// ------------------------------------------------------------------ //
// Section 0 -- cursor baseline, and the enable/disable edges.
// ------------------------------------------------------------------ //

// First time we ever run, adopt whatever the ring can still supply rather than
// starting at nWriteIdx. Someone who enables logging after noticing trouble
// wants the entries that are still there, not only the ones from now on. Bounded
// by RING because older slots have already been overwritten.
IF NOT bCursorSet THEN
    bCursorSet := TRUE;
    IF GVL_Log.nWriteIdx > RING THEN
        udiLastRead := GVL_Log.nWriteIdx - RING;
    ELSE
        udiLastRead := 0;
    END_IF
END_IF

// Turning logging OFF must not abandon a part-written flush or a full buffer:
// drain what is pending and close cleanly, THEN go idle.
fbTrigOff(CLK := NOT GVL_HmiPersistent.stLogFileCfg.bEnabled);
IF fbTrigOff.Q AND (GVL_Log.nWriteIdx > udiLastRead) THEN
    bClosing := TRUE;
END_IF

udiPending := GVL_Log.nWriteIdx - udiLastRead;

// ------------------------------------------------------------------ //
// Section 1 -- flush trigger.
//
// The quiet timer is the flash-wear control: entries collect in the ring and
// reach the card once per uiFlushSec, so a busy second costs one open/close
// rather than dozens. HIGH_WATER is the safety valve -- at 200 of 256 pending
// we stop waiting for the timer, because passing 256 loses entries.
// ------------------------------------------------------------------ //
tonFlush(IN  := (udiPending > 0) AND GVL_HmiPersistent.stLogFileCfg.bEnabled,
         PT  := UDINT_TO_TIME(GVL_HmiPersistent.stLogFileCfg.uiFlushSec * 1000));

// ------------------------------------------------------------------ //
// Section 2 -- the state machine.
// ------------------------------------------------------------------ //
CASE eStep OF

// ---------------- 0: idle ---------------- //
0:
    // OFF means "not logging". BUFFER means "logging, entries accumulating in the
    // ring, waiting for the flush interval". Reporting OFF while enabled would
    // read as a fault on the Logs page when nothing is wrong.
    IF GVL_HmiPersistent.stLogFileCfg.bEnabled THEN
        GVL_Log.stLogFile.eState := E_LogFileState.BUFFER;
    ELSE
        GVL_Log.stLogFile.eState := E_LogFileState.OFF;
    END_IF

    IF (GVL_HmiPersistent.stLogFileCfg.bEnabled OR bClosing)
       AND (udiPending > 0)
       AND (tonFlush.Q OR (udiPending >= HIGH_WATER) OR bClosing) THEN

        // OVERFLOW CHECK, before anything else touches the cursor. If more than
        // RING entries arrived since we last read, the oldest are already
        // overwritten and are gone -- unavoidable, the ring is finite. What is
        // NOT acceptable is losing them silently, so the count is published AND
        // a synthetic row goes into the file itself. A reader of the CSV must be
        // able to see the gap without also having to read a PLC symbol.
        IF udiPending > RING THEN
            udiLostNow := udiPending - RING;
            GVL_Log.stLogFile.udiEntriesDropped :=
                GVL_Log.stLogFile.udiEntriesDropped + udiLostNow;
            udiLastRead := GVL_Log.nWriteIdx - RING;
            bLossRow    := TRUE;
        END_IF

        GVL_Log.stLogFile.eState := E_LogFileState.BUFFER;
        eStep := 5;
    END_IF

// ---------------- 5: make sure the directory exists ---------------- //
// Once per session. Errors are IGNORED on purpose: "already exists" is an error
// from this FB and is also the normal case, and distinguishing it from a real
// failure by error number would be guessing. If the directory genuinely cannot
// be made, the open in state 20 fails and THAT is reported -- one authoritative
// error rather than two competing ones.
5:
    IF bDirTried THEN
        eStep := 10;
    ELSE
        sDirNoSlash := GVL_HmiPersistent.stLogFileCfg.sDir;
        IF (LEN(sDirNoSlash) > 1)
           AND (RIGHT(sDirNoSlash, 1) = '\') THEN
            sDirNoSlash := LEFT(sDirNoSlash, LEN(sDirNoSlash) - 1);
        END_IF
        fbMkDir(sPathName := sDirNoSlash,
                ePath     := Tc2_System.PATH_GENERIC,
                bExecute  := TRUE,
                tTimeout  := FILE_TO);
        IF NOT fbMkDir.bBusy THEN
            fbMkDir(bExecute := FALSE);
            bDirTried := TRUE;
            eStep := 10;
        END_IF
    END_IF

// ---------------- 10: filename, and does it already exist? ---------------- //
10:
    IF GVL_Log.sToday = '0000-00-00' THEN
        // The panel RTC is unset. Naming a file from that would produce
        // something like flower-0000-00-00.csv, which sorts before every real
        // file and would be deleted first by the Phase 3 retention sweep -- so
        // the one file written while the clock was broken would be the first to
        // go. A distinct name keeps it identifiable and out of the date order.
        sFileName := 'flower-nodate.csv';
    ELSE
        sFileName := CONCAT(CONCAT('flower-', GVL_Log.sToday), '.csv');
    END_IF
    sPath := CONCAT(GVL_HmiPersistent.stLogFileCfg.sDir, sFileName);

    IF sFileName = sLastFile THEN
        bNeedHeader := FALSE;       // same file we appended to last time
        eStep := 20;
    ELSE
        eStep := 11;                // new name -- has to be tested
    END_IF

// ---------------- 11/12: existence probe ---------------- //
// A header belongs at the top of a file, once. Opening in append mode cannot
// tell us whether we created it, so we test first with a READ open: 1804 means
// absent, which is the one error code this project has verified on the panel.
// Costs one extra call per new file, i.e. once a day.
11:
    fbProbe(sPathName := sPath,
            nMode     := Tc2_System.FOPEN_MODEREAD,
            ePath     := Tc2_System.PATH_GENERIC,
            bExecute  := TRUE,
            tTimeout  := FILE_TO);
    IF NOT fbProbe.bBusy THEN
        fbProbe(bExecute := FALSE);
        IF fbProbe.bError THEN
            // Absent -> new file, needs a header. Any OTHER error is left for
            // the append open in state 20 to report, so there is one place that
            // decides the directory is unusable.
            bNeedHeader := (fbProbe.nErrId = E_NOTFOUND);
            eStep := 20;
        ELSE
            bNeedHeader := FALSE;
            hFile := fbProbe.hFile;
            eStep := 12;            // must close the probe handle
        END_IF
    END_IF

12:
    fbClose(hFile := hFile, bExecute := TRUE, tTimeout := FILE_TO);
    IF NOT fbClose.bBusy THEN
        fbClose(bExecute := FALSE);
        hFile := 0;
        eStep := 20;
    END_IF

// ---------------- 20: open for append ---------------- //
20:
    GVL_Log.stLogFile.eState := E_LogFileState.OPENING;
    fbOpen(sPathName := sPath,
           nMode     := Tc2_System.FOPEN_MODEAPPEND OR Tc2_System.FOPEN_MODETEXT,
           ePath     := Tc2_System.PATH_GENERIC,
           bExecute  := TRUE,
           tTimeout  := FILE_TO);
    IF NOT fbOpen.bBusy THEN
        fbOpen(bExecute := FALSE);
        IF fbOpen.bError THEN
            Fail(nErr := fbOpen.nErrId, sWhy := 'open failed');
        ELSE
            hFile := fbOpen.hFile;
            IF bNeedHeader THEN
                sLastFile := sFileName;
                GVL_Log.stLogFile.sCurrentFile := sFileName;
                GVL_Log.stLogFile.uiBytesInFile := 0;
                eStep := 25;
            ELSE
                sLastFile := sFileName;
                GVL_Log.stLogFile.sCurrentFile := sFileName;
                eStep := 30;
            END_IF
        END_IF
    END_IF

// ---------------- 25: header row, new files only ---------------- //
25:
    GVL_Log.stLogFile.eState := E_LogFileState.WRITING;
    fbPuts(hFile := hFile, sLine := CONCAT(HDR, '$N'),
           bExecute := TRUE, tTimeout := FILE_TO);
    IF NOT fbPuts.bBusy THEN
        fbPuts(bExecute := FALSE);
        IF fbPuts.bError THEN
            Fail(nErr := fbPuts.nErrId, sWhy := 'header write failed');
        ELSE
            // +1 because text mode expands the single $N to CRLF on disk.
            GVL_Log.stLogFile.uiBytesInFile :=
                GVL_Log.stLogFile.uiBytesInFile + INT_TO_UDINT(LEN(HDR)) + 2;
            bNeedHeader := FALSE;
            eStep := 30;
        END_IF
    END_IF

// ---------------- 30: the synthetic loss row, if one is owed ---------------- //
30:
    IF NOT bLossRow THEN
        eStep := 31;
    ELSE
        GVL_Log.stLogFile.eState := E_LogFileState.WRITING;
        sRow := CONCAT(CONCAT(Csv(sIn := GVL_Log.sNow), ',"WARN","LogCsv","'),
                CONCAT(UDINT_TO_STRING(udiLostNow),
                       ' entries lost - CSV writer fell behind the ring"$N'));
        fbPuts(hFile := hFile, sLine := sRow,
               bExecute := TRUE, tTimeout := FILE_TO);
        IF NOT fbPuts.bBusy THEN
            fbPuts(bExecute := FALSE);
            IF fbPuts.bError THEN
                Fail(nErr := fbPuts.nErrId, sWhy := 'loss row write failed');
            ELSE
                GVL_Log.stLogFile.uiBytesInFile :=
                    GVL_Log.stLogFile.uiBytesInFile + INT_TO_UDINT(LEN(sRow)) + 1;
                bLossRow := FALSE;
                eStep := 31;
            END_IF
        END_IF
    END_IF

// ---------------- 31: one row per pass until caught up ---------------- //
31:
    IF udiLastRead >= GVL_Log.nWriteIdx THEN
        eStep := 40;
    ELSE
        // Discard DBG without a file call. Unconditional -- independent of
        // GVL_Log.bDebugMode, which still governs the on-screen ring. DBG is the
        // 1 Hz robot keep-alive trace; it would bury the file and burn the card.
        // Bounded per scan so a long DBG run cannot stretch the PlcTask.
        nSkipped := 0;
        WHILE (udiLastRead < GVL_Log.nWriteIdx)
              AND (nSkipped < MAX_SKIP) DO
            nSlot := UDINT_TO_INT(udiLastRead MOD RING);
            IF GVL_Log.aLog[nSlot].eSev = E_LogSev.DBG THEN
                udiLastRead := udiLastRead + 1;
                nSkipped := nSkipped + 1;
            ELSE
                EXIT;
            END_IF
        END_WHILE

        IF udiLastRead >= GVL_Log.nWriteIdx THEN
            eStep := 40;
        ELSE
            GVL_Log.stLogFile.eState := E_LogFileState.WRITING;
            nSlot := UDINT_TO_INT(udiLastRead MOD RING);
            sRow  := RowFor(nSlot := nSlot);
            fbPuts(hFile := hFile, sLine := sRow,
                   bExecute := TRUE, tTimeout := FILE_TO);
            IF NOT fbPuts.bBusy THEN
                fbPuts(bExecute := FALSE);
                IF fbPuts.bError THEN
                    Fail(nErr := fbPuts.nErrId, sWhy := 'row write failed');
                ELSE
                    // Cursor advances ONLY after the write is confirmed. If it
                    // advanced first, a failure here would drop the entry
                    // permanently and invisibly -- the one outcome this whole FB
                    // is arranged to prevent.
                    udiLastRead := udiLastRead + 1;
                    GVL_Log.stLogFile.uiBytesInFile :=
                        GVL_Log.stLogFile.uiBytesInFile + INT_TO_UDINT(LEN(sRow)) + 1;
                END_IF
            END_IF
        END_IF
    END_IF

// ---------------- 40: close ---------------- //
40:
    GVL_Log.stLogFile.eState := E_LogFileState.CLOSING;
    fbClose(hFile := hFile, bExecute := TRUE, tTimeout := FILE_TO);
    IF NOT fbClose.bBusy THEN
        fbClose(bExecute := FALSE);
        IF fbClose.bError THEN
            Fail(nErr := fbClose.nErrId, sWhy := 'close failed');
        ELSE
            hFile := 0;
            // One INFO out, matching the one ERR in. Same discipline as
            // FB_RobotTcpClient's bStateUnanswered: a repeating condition must
            // not be level-logged into a 20-entry ring.
            IF bErrLogged THEN
                bErrLogged := FALSE;
                GVL_Log.stLogFile.iErrorCode := 0;
                GVL_Log.stLogFile.sErrorText := '';
                F_LogEvent(eSev := E_LogSev.INFO, sSource := 'LogCsv',
                           sMsg  := CONCAT('CSV log recovered, writing ',
                                           sFileName));
            END_IF
            tonFlush(IN := FALSE);      // restart the quiet interval
            bClosing := FALSE;
            eStep := 0;
        END_IF
    END_IF

// ---------------- 90: release the handle on the way to FAILED ---------------- //
// Reached only from Fail() and only when a handle is still open. The close result
// is IGNORED: we are already reporting the original error, and replacing it with
// a close error would lose the diagnosis that matters. What we need from here is
// the handle back, not a second opinion.
90:
    GVL_Log.stLogFile.eState := E_LogFileState.CLOSING;
    fbClose(hFile := hFile, bExecute := TRUE, tTimeout := FILE_TO);
    IF NOT fbClose.bBusy THEN
        fbClose(bExecute := FALSE);
        hFile := 0;
        eStep := 99;
    END_IF

// ---------------- 99: failed -- back off, then retry ---------------- //
// Retry on a TIMER, never every scan. A bad sDir or a full card would otherwise
// produce a file call per scan for as long as the machine runs.
99:
    GVL_Log.stLogFile.eState := E_LogFileState.FAILED;
    tonRetry(IN := TRUE, PT := RETRY_TO);
    IF tonRetry.Q THEN
        tonRetry(IN := FALSE);
        bDirTried := FALSE;             // maybe the card came back
        sLastFile := '';                // re-test existence
        eStep := 0;
    END_IF

END_CASE

// ------------------------------------------------------------------ //
// Section 3 -- the STRING mirror of eState.
//
// Required, not decoration: the classic VISU cannot stringify an enum, so a text
// output bound to eState renders the raw number. Every enum in this project
// carries such a mirror for that reason.
// ------------------------------------------------------------------ //
CASE GVL_Log.stLogFile.eState OF
    E_LogFileState.OFF:      GVL_Log.stLogFile.sStateText := 'OFF';
    E_LogFileState.BUFFER:   GVL_Log.stLogFile.sStateText := 'BUFFER';
    E_LogFileState.OPENING:  GVL_Log.stLogFile.sStateText := 'OPENING';
    E_LogFileState.WRITING:  GVL_Log.stLogFile.sStateText := 'WRITING';
    E_LogFileState.CLOSING:  GVL_Log.stLogFile.sStateText := 'CLOSING';
    E_LogFileState.ROTATING: GVL_Log.stLogFile.sStateText := 'ROTATING';
    E_LogFileState.FAILED:   GVL_Log.stLogFile.sStateText := 'FAILED';
ELSE
    GVL_Log.stLogFile.sStateText := '?';
END_CASE

(*
   RFC 4180 quote one field: wrap in double quotes, and double any quote inside.

   NOT theoretical. Robot frames reach log messages as 'SYNC:NAME=VALUE,...' and
   message text already carries commas and parentheses, so an unquoted field
   would split a row into the wrong number of columns and silently corrupt every
   downstream reader. Verified end-to-end on the panel 2026-08-10: a message
   containing both a comma and a doubled quote came back off the card via FTP and
   parsed as one intact field.

   Every field is quoted, including the fixed ones. Uniform rows are easier to
   reason about than rows where quoting depends on content, and the cost is two
   bytes.
*)
METHOD Csv : STRING(200)
VAR_INPUT
    sIn : STRING(80);
END_VAR
VAR
    j    : INT;
    n    : INT;
    sOut : STRING(200);
    c    : STRING(1);
END_VAR
sOut := '"';
n := LEN(sIn);

FOR j := 1 TO n DO
    c := MID(sIn, 1, j);            // MID(str, len, pos) -- one char at j
    IF c = '"' THEN
        sOut := CONCAT(sOut, '""');
    ELSE
        sOut := CONCAT(sOut, c);
    END_IF
END_FOR

Csv := CONCAT(sOut, '"');
END_METHOD

(*
   Build one CSV row from a ring slot, ending in a bare $N.

   Column order matches the HDR constant. Worst case fits: the four source
   fields are STRING(8), STRING(8), STRING(20) and STRING(80), so fully
   quote-doubled they come to 18 + 18 + 42 + 162, plus three commas and the
   newline = 244 of the 255 available.

   $N and NOT $R$N -- FOPEN_MODETEXT already produces CRLF, and doubling it
   gives \r\r\n. See the FB header.
*)
METHOD RowFor : STRING(255)
VAR_INPUT
    nSlot : INT;
END_VAR
RowFor := CONCAT(Csv(sIn := GVL_Log.aLog[nSlot].sTime), ',');
RowFor := CONCAT(RowFor, CONCAT(Csv(sIn := GVL_Log.aLog[nSlot].sSevText), ','));
RowFor := CONCAT(RowFor, CONCAT(Csv(sIn := GVL_Log.aLog[nSlot].sSource), ','));
RowFor := CONCAT(RowFor, CONCAT(Csv(sIn := GVL_Log.aLog[nSlot].sMsg), '$N'));
END_METHOD

(*
   One place that gives up on a flush: latch the error, release the handle, log
   once, and drop into the backoff state.

   THE LOG IS EDGE-GUARDED, and that is the point of centralising this. A full
   card or a bad sDir repeats every retry interval, and level-logging it would
   flush the 20-entry aRecent ring and hide whatever caused the trouble --
   exactly the defect this project already has open against
   FB_RobotTcpClient's connect-failure path. One ERR in, one INFO out on
   recovery (state 40).

   IT DOES NOT CLOSE THE HANDLE ITSELF. An earlier version did, with one
   bExecute TRUE/FALSE pair in the same scan, which starts the close and disarms
   it before it can finish -- so the handle leaks. Harmless once; but a failure
   that repeats every RETRY_TO leaks one every 30 s for as long as the machine
   runs, and exhausting the runtime's handle table would then present as the file
   blocks having stopped working. So a still-open handle routes through state 90,
   which closes it asynchronously and properly before the backoff.
*)
METHOD Fail : BOOL
VAR_INPUT
    nErr : UDINT;
    sWhy : STRING(40);
END_VAR
GVL_Log.stLogFile.iErrorCode := nErr;
GVL_Log.stLogFile.sErrorText :=
    CONCAT(CONCAT(sWhy, ' err '), UDINT_TO_STRING(nErr));

IF NOT bErrLogged THEN
    bErrLogged := TRUE;
    F_LogEvent(eSev := E_LogSev.ERR, sSource := 'LogCsv',
               sMsg  := CONCAT(CONCAT(GVL_Log.stLogFile.sErrorText, ' ('),
                               CONCAT(sPath, ')')));
END_IF

bClosing := FALSE;

// A handle we opened is still open -- close it properly first (state 90) rather
// than abandoning it. See the header: abandoning leaks one handle per retry.
IF hFile <> 0 THEN
    eStep := 90;
ELSE
    eStep := 99;
END_IF

Fail := TRUE;
END_METHOD

END_FUNCTION_BLOCK

// ---- POUs/FB_SolSolPiston_2Pos.TcPOU
FUNCTION_BLOCK FB_SolSolPiston_2Pos
VAR_INPUT
    (* Automatic Commands from PLC sequence logic. Wired to FALSE in MAIN until FB_Auto exists. *)
    bAutoCmdExtend    : BOOL;
    bAutoCmdRetract   : BOOL;

    (* Physical Feedback (Proximity Switches) *)
    bSwitchExtended   : BOOL;
    bSwitchRetracted  : BOOL;
END_VAR

VAR_IN_OUT
    (* HMI contract — mode, manual + simulate inputs, latched + sensor status *)
    stHmi             : ST_HmiPiston;
END_VAR

VAR_OUTPUT
    (* Physical Outputs to Solenoids *)
    bOutSolenoidExtend  : BOOL;
    bOutSolenoidRetract : BOOL;
END_VAR

VAR
    (* Internal Target States *)
    bTargetExtend     : BOOL;
    bTargetRetract    : BOOL;

    (* HMI Manual-Button Edge Detection *)
    fbTrigManExtend   : R_TRIG;
    fbTrigManRetract  : R_TRIG;

    (* Effective sensor states = real OR HMI simulate. Recomputed every cycle in Section 0a. *)
    bSwitchExtended_eff  : BOOL;
    bSwitchRetracted_eff : BOOL;

    (* Previous-cycle snapshots for the mode-field bridge in Section 0b.
       Classic PLC HMI writes stHmi.bMode (Rotary Switch is boolean-only);
       web HMI writes stHmi.eMode (enum via ToggleSwitch). This FB is the
       authoritative reader of eMode, so we sync in whichever direction
       changed since last cycle. *)
    bPrevMode : BOOL;
    ePrevMode : E_ControlMode;
END_VAR

(* ==========================================
   0b. MODE-FIELD BRIDGE — sync bMode <-> eMode
   The classic PLC HMI (VISUs) writes stHmi.bMode because its Rotary Switch
   element is boolean-only. FlowerPyHmi writes stHmi.eMode over ADS.
   (The retired Flower_HMI web project did the same via a ToggleSwitch.) Rest of this FB reads eMode as the authoritative field,
   so we mirror bMode into eMode when the classic HMI toggled the switch,
   and mirror eMode back into bMode when the web HMI (or anyone else) wrote
   eMode. Edge-triggered — whichever side changed since last cycle wins.
   Runs BEFORE Section 0 so downstream logic sees a coherent eMode.
   ========================================== *)
IF stHmi.bMode <> bPrevMode THEN
    // Classic VISU changed bMode → propagate to eMode
    IF stHmi.bMode THEN
        stHmi.eMode := E_ControlMode.Automatic;
    ELSE
        stHmi.eMode := E_ControlMode.Manual;
    END_IF;
ELSIF stHmi.eMode <> ePrevMode THEN
    // Web HMI (or any other writer) changed eMode → propagate to bMode
    stHmi.bMode := (stHmi.eMode = E_ControlMode.Automatic);
END_IF;

bPrevMode := stHmi.bMode;
ePrevMode := stHmi.eMode;

(* ==========================================
   0a. EFFECTIVE SENSOR INPUTS (real OR HMI simulate)
   ========================================== *)
bSwitchExtended_eff  := bSwitchExtended  OR stHmi.bSimulateExtended;
bSwitchRetracted_eff := bSwitchRetracted OR stHmi.bSimulateRetracted;

(* ==========================================
   0. HMI MANUAL BUTTON LATCHING (Radio-Button Behavior)
   ========================================== *)
fbTrigManExtend(CLK := stHmi.bManCmdExtend);
fbTrigManRetract(CLK := stHmi.bManCmdRetract);

// Independent IFs (not ELSIF): if multiple edges fire in the same cycle, the last one wins (Retract > Extend).
IF fbTrigManExtend.Q  THEN stHmi.bSelectedExtend := TRUE;  stHmi.bSelectedRetract := FALSE; END_IF;
IF fbTrigManRetract.Q THEN stHmi.bSelectedExtend := FALSE; stHmi.bSelectedRetract := TRUE;  END_IF;

IF stHmi.eMode = E_ControlMode.Automatic THEN
    stHmi.bSelectedExtend := FALSE; stHmi.bSelectedRetract := FALSE;
END_IF;

(* ==========================================
   1. MODE SELECTION & COMMAND MAPPING
   ========================================== *)
IF stHmi.eMode = E_ControlMode.Automatic THEN
    bTargetExtend  := bAutoCmdExtend;
    bTargetRetract := bAutoCmdRetract;

ELSIF stHmi.eMode = E_ControlMode.Manual THEN
    bTargetExtend  := stHmi.bSelectedExtend;
    bTargetRetract := stHmi.bSelectedRetract;

ELSE
    // Safe default: undefined mode → no targets
    bTargetExtend  := FALSE;
    bTargetRetract := FALSE;
END_IF;

(* ==========================================
   1a. JOG OVERRIDE — clear latched selection while either jog is held
   ========================================== *)
// Section 1 above already copied stHmi.bSelected* into bTarget*. The stale
// bTarget* is harmless because Section 2's jog branches sit ahead of the
// bTarget* branches in the IF/ELSIF ladder and preempt them.
IF stHmi.bManJogExtend OR stHmi.bManJogRetract THEN
    stHmi.bSelectedExtend := FALSE; stHmi.bSelectedRetract := FALSE;
END_IF;

(* ==========================================
   1b. TARGET-REACHED RESET — clear bSelected* once the piston arrives
   ========================================== *)
IF stHmi.bSelectedExtend  AND bSwitchExtended_eff  THEN stHmi.bSelectedExtend  := FALSE; END_IF;
IF stHmi.bSelectedRetract AND bSwitchRetracted_eff THEN stHmi.bSelectedRetract := FALSE; END_IF;

(* ==========================================
   2. SOLENOID CONTROL — Jog takes priority over latched target
   ========================================== *)
// Jog branches first, gated by Manual mode. If both jogs are held
// simultaneously, Retract wins (matching the same-cycle collision rule
// in Section 0). Each branch still respects the corresponding effective
// sensor. In Automatic mode the jog branches are skipped entirely so
// bAutoCmd* controls the piston.

// JOG EXTEND: while held in Manual, drive Extend coil until end sensor
IF stHmi.bManJogExtend AND NOT bSwitchExtended_eff AND stHmi.eMode = E_ControlMode.Manual THEN
    bOutSolenoidExtend  := TRUE;
    bOutSolenoidRetract := FALSE;

// JOG RETRACT: while held in Manual, drive Retract coil until end sensor
ELSIF stHmi.bManJogRetract AND NOT bSwitchRetracted_eff AND stHmi.eMode = E_ControlMode.Manual THEN
    bOutSolenoidRetract := TRUE;
    bOutSolenoidExtend  := FALSE;

// CASE 1: Move to EXTENDED position (latched target)
ELSIF bTargetExtend AND NOT bSwitchExtended_eff THEN
    bOutSolenoidExtend  := TRUE;
    bOutSolenoidRetract := FALSE;

// CASE 2: Move to RETRACTED position (latched target)
ELSIF bTargetRetract AND NOT bSwitchRetracted_eff THEN
    bOutSolenoidRetract := TRUE;
    bOutSolenoidExtend  := FALSE;

// CASE 3: Target reached or no active target → stop both coils
ELSE
    bOutSolenoidExtend  := FALSE;
    bOutSolenoidRetract := FALSE;
END_IF;

(* ==========================================
   3. HMI STATUS FEEDBACK
   ========================================== *)
stHmi.bIsExtended        := bSwitchExtended_eff;
stHmi.bIsRetracted       := bSwitchRetracted_eff;
stHmi.bIsMoving          := bOutSolenoidExtend OR bOutSolenoidRetract;
stHmi.bOutSolenoidExtend  := bOutSolenoidExtend;
stHmi.bOutSolenoidRetract := bOutSolenoidRetract;

END_FUNCTION_BLOCK

// ---- GlobalTextList.TcGTLO
TEXTLIST GlobalTextList
  72 = '%s'
  899 = 'Auto'
  1020 = 'Auto Main'
  1107 = 'Auto Mode'
  593 = 'Auto/Man'
  658 = 'Auto/Manual'
  1021 = 'Back'
  841 = 'bManCmdExtend'
  294 = 'bManCmdRetract'
  296 = 'bManJogExtend'
  926 = 'bManJogRetract'
  1106 = 'START'
  923 = 'Main'
  57 = 'Man'
  58 = 'MOVING'
  1108 = 'No sensors (timed steps)'
  551 = 'Gripper Manual'
  650 = 'PB1 hold STOP (ms)'
  651 = 'PB2+PB3 hold (ms)'
  600 = 'Robot'
  601 = 'Connection'
  602 = '%s'
  603 = 'Packets Rx'
  604 = '%d'
  605 = 'Packets Tx'
  606 = '%d'
  607 = 'Last Rx'
  608 = '%s'
  609 = 'Last Tx'
  610 = '%s'
  611 = 'State out'
  612 = '%d'
  613 = 'Robot cmd'
  614 = '%d'
  615 = 'Get Sync'
  616 = 'New Bulb'
  552 = 'Robot'
  620 = 'J_SPEED'
  621 = 'L_SPEED'
  622 = 'REPEATS'
  623 = 'START_WAIT'
  624 = 'WATER_WAIT'
  625 = 'STAND_WAIT'
  626 = 'END_WAIT'
  627 = 'WATER_SPEED'
  628 = 'WAX_WAIT_TIME_IN'
  629 = 'WAX_WAIT_TIME_OUT'
  630 = 'WAX_SPEED'
  640 = 'tDwellPushMs'
  641 = 'tPushRetractedDwellMs'
  642 = 'tSepRetractedDwellMs'
  643 = 'tStepTimeoutMs'
  644 = 'tPlateWaitTimeoutMs'
  660 = 'Bypass plate sensors'
  670 = 'Plate'
  671 = 'L'
  672 = 'R'
  1200 = 'Log'
  1201 = 'Enabled'
  1202 = 'Debug'
  1203 = 'Writes'
  1204 = '%d'
  1205 = 'Sev'
  1206 = 'Time'
  1207 = 'Message'
  1208 = '%s'
  1209 = '%s'
  1210 = '%s'
  1211 = '%s'
  1212 = '%s'
  1213 = '%s'
  1214 = '%s'
  1215 = '%s'
  1216 = '%s'
  1217 = '%s'
  1218 = '%s'
  1219 = '%s'
  1220 = '%s'
  1221 = '%s'
  1222 = '%s'
  1223 = '%s'
  1224 = '%s'
  1225 = '%s'
  1226 = '%s'
  1227 = '%s'
  1228 = '%s'
  1229 = '%s'
  1230 = '%s'
  1231 = '%s'
  1232 = '%s'
  1233 = '%s'
  1234 = '%s'
  1235 = '%s'
  1236 = '%s'
  1237 = '%s'
  1238 = '%s'
  1239 = '%s'
  1240 = '%s'
  1241 = '%s'
  1242 = '%s'
  1243 = '%s'
  1244 = '%s'
  1245 = '%s'
  1246 = '%s'
  1247 = '%s'
  1248 = '%s'
  1249 = '%s'
  1250 = '%s'
  1251 = '%s'
  1252 = '%s'
  1253 = '%s'
  1254 = '%s'
  1255 = '%s'
  1256 = '%s'
  1257 = '%s'
  1258 = '%s'
  1259 = '%s'
  1260 = '%s'
  1261 = '%s'
  1262 = '%s'
  1263 = '%s'
  1264 = '%s'
  1265 = '%s'
  1266 = '%s'
  1267 = '%s'
  1199 = 'Log'
  1300 = 'Robot IP'
  1301 = '%s'
  1100 = 'Auto Config'
  1302 = 'Back'
  1303 = 'Auto Config'
  1304 = 'File log'
  1305 = 'Failed connects'
  550 = 'Pistons Manual'
  1105 = 'RESET'
  429 = 'SimEXT'
  52 = 'SimRET'
  1103 = 'ENABLE AUTO'
  1104 = 'STOP'
END_TEXTLIST

// ---- VISU/Main.TcVIS
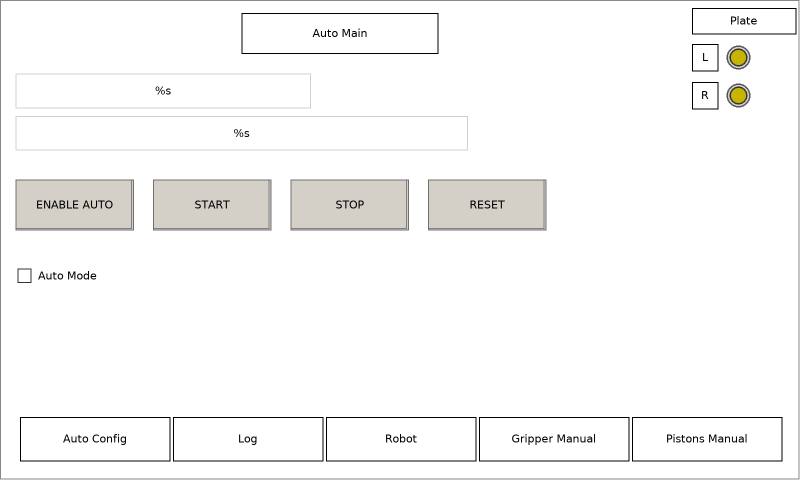
VISUALIZATION Main  // 800x480
    Rectangle (632,417 150x44), "Pistons Manual"
        OnMouseDown: change screen: PistonsManual
    Rectangle (326,417 150x44), "Robot"
        OnMouseDown: change screen: Robot
    Rectangle (173,417 150x44), "Log"
        OnMouseDown: change screen: Logs
    Rectangle (479,417 150x44), "Gripper Manual"
        OnMouseDown: change screen: GripperManual
    Frame (-4,3 688x404)
        shows AutoMain(stMasterAutoCycle := GVL_HMI.stMasterAuto, stCfg := GVL_HmiPersistent.stMasterAutoCfg)
    Rectangle (692,8 104x26), "Plate"
    Rectangle (692,44 26x27), "L"
    Lamp1 (724,44 29x27), variable: GVL_HMI.bPlateSenL, style: Lamp-Lamp1-Yellow
    Rectangle (692,82 26x27), "R"
    Lamp1 (724,82 29x27), variable: GVL_HMI.bPlateSenR, style: Lamp-Lamp1-Yellow
    Rectangle (20,417 150x44), "Auto Config"
        OnMouseDown: change screen: AutoConfig
END_VISUALIZATION

// ---- VISU/PistonsManual.TcVIS
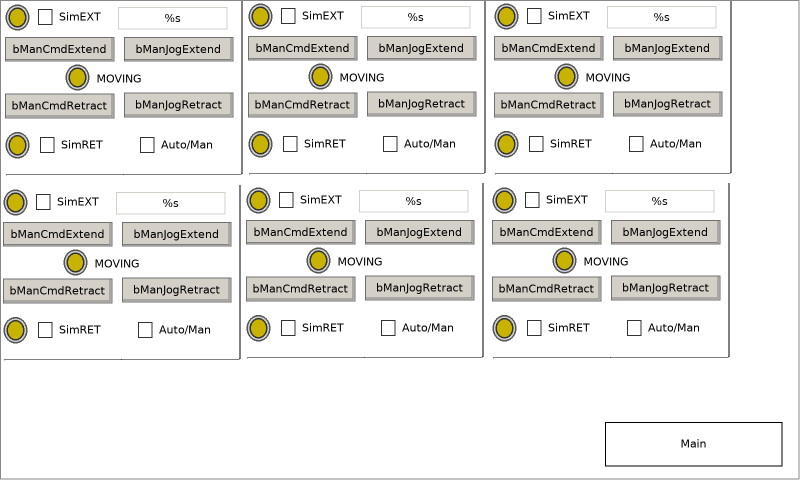
VISUALIZATION PistonsManual  // 800x480
    Frame (-3,-3 250x200)
        shows Piston(piston := GVL_HMI.stSepSol1)
    Rectangle (605,422 177x44), "Main"
        OnMouseDown: change screen: Main
    Frame (-5,182 250x200)
        shows Piston(piston := GVL_HMI.stPushSol1)
    Frame (240,-4 250x200)
        shows Piston(piston := GVL_HMI.stSepSol2)
    Frame (238,180 250x200)
        shows Piston(piston := GVL_HMI.stPushSol2)
    Frame (486,-4 250x200)
        shows Piston(piston := GVL_HMI.stSepSol3)
    Frame (484,180 250x200)
        shows Piston(piston := GVL_HMI.stPushSol3)
END_VISUALIZATION

// ---- VISU/Logs.TcVIS
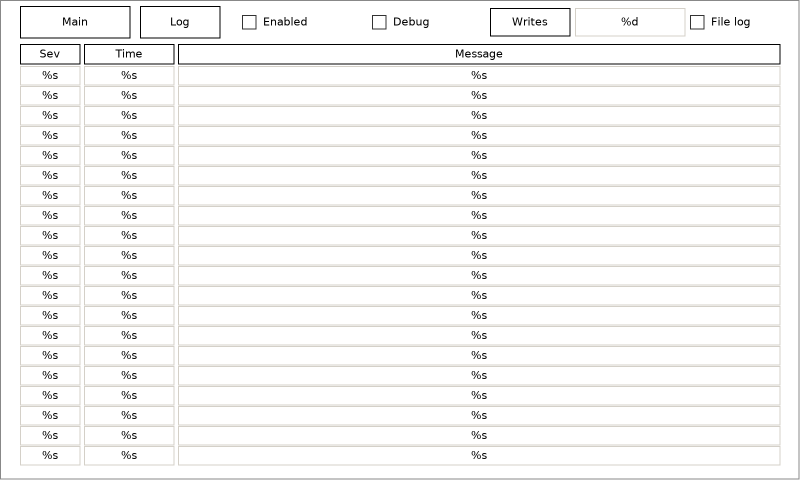
VISUALIZATION Logs  // 800x480
    Rectangle (20,6 110x32), "Main"
        OnMouseDown: change screen: Main
    Rectangle (140,6 80x32), "Log"
    Checkbox (240,8 120x28), "Enabled", variable: GVL_Log.bLogEnabled
    Checkbox (370,8 110x28), "Debug", variable: GVL_Log.bDebugMode
    Checkbox (688,8 110x28), "File log", variable: GVL_HmiPersistent.stLogFileCfg.bEnabled
    Rectangle (490,8 80x28), "Writes"
    Textfield (575,8 110x28), "%d", text variable: GVL_Log.nWriteIdx
    Rectangle (20,44 60x20), "Sev"
    Rectangle (84,44 90x20), "Time"
    Rectangle (178,44 602x20), "Message"
    Textfield (20,66 60x19), "%s", text variable: GVL_Log.aRecent[0].sSevText
    Textfield (84,66 90x19), "%s", text variable: GVL_Log.aRecent[0].sTime
    Textfield (178,66 602x19), "%s", text variable: GVL_Log.aRecent[0].sMsg
    Textfield (20,86 60x19), "%s", text variable: GVL_Log.aRecent[1].sSevText
    Textfield (84,86 90x19), "%s", text variable: GVL_Log.aRecent[1].sTime
    Textfield (178,86 602x19), "%s", text variable: GVL_Log.aRecent[1].sMsg
    Textfield (20,106 60x19), "%s", text variable: GVL_Log.aRecent[2].sSevText
    Textfield (84,106 90x19), "%s", text variable: GVL_Log.aRecent[2].sTime
    Textfield (178,106 602x19), "%s", text variable: GVL_Log.aRecent[2].sMsg
    Textfield (20,126 60x19), "%s", text variable: GVL_Log.aRecent[3].sSevText
    Textfield (84,126 90x19), "%s", text variable: GVL_Log.aRecent[3].sTime
    Textfield (178,126 602x19), "%s", text variable: GVL_Log.aRecent[3].sMsg
    Textfield (20,146 60x19), "%s", text variable: GVL_Log.aRecent[4].sSevText
    Textfield (84,146 90x19), "%s", text variable: GVL_Log.aRecent[4].sTime
    Textfield (178,146 602x19), "%s", text variable: GVL_Log.aRecent[4].sMsg
    Textfield (20,166 60x19), "%s", text variable: GVL_Log.aRecent[5].sSevText
    Textfield (84,166 90x19), "%s", text variable: GVL_Log.aRecent[5].sTime
    Textfield (178,166 602x19), "%s", text variable: GVL_Log.aRecent[5].sMsg
    Textfield (20,186 60x19), "%s", text variable: GVL_Log.aRecent[6].sSevText
    Textfield (84,186 90x19), "%s", text variable: GVL_Log.aRecent[6].sTime
    Textfield (178,186 602x19), "%s", text variable: GVL_Log.aRecent[6].sMsg
    Textfield (20,206 60x19), "%s", text variable: GVL_Log.aRecent[7].sSevText
    Textfield (84,206 90x19), "%s", text variable: GVL_Log.aRecent[7].sTime
    Textfield (178,206 602x19), "%s", text variable: GVL_Log.aRecent[7].sMsg
    Textfield (20,226 60x19), "%s", text variable: GVL_Log.aRecent[8].sSevText
    Textfield (84,226 90x19), "%s", text variable: GVL_Log.aRecent[8].sTime
    Textfield (178,226 602x19), "%s", text variable: GVL_Log.aRecent[8].sMsg
    Textfield (20,246 60x19), "%s", text variable: GVL_Log.aRecent[9].sSevText
    Textfield (84,246 90x19), "%s", text variable: GVL_Log.aRecent[9].sTime
    Textfield (178,246 602x19), "%s", text variable: GVL_Log.aRecent[9].sMsg
    Textfield (20,266 60x19), "%s", text variable: GVL_Log.aRecent[10].sSevText
    Textfield (84,266 90x19), "%s", text variable: GVL_Log.aRecent[10].sTime
    Textfield (178,266 602x19), "%s", text variable: GVL_Log.aRecent[10].sMsg
    Textfield (20,286 60x19), "%s", text variable: GVL_Log.aRecent[11].sSevText
    Textfield (84,286 90x19), "%s", text variable: GVL_Log.aRecent[11].sTime
    Textfield (178,286 602x19), "%s", text variable: GVL_Log.aRecent[11].sMsg
    Textfield (20,306 60x19), "%s", text variable: GVL_Log.aRecent[12].sSevText
    Textfield (84,306 90x19), "%s", text variable: GVL_Log.aRecent[12].sTime
    Textfield (178,306 602x19), "%s", text variable: GVL_Log.aRecent[12].sMsg
    Textfield (20,326 60x19), "%s", text variable: GVL_Log.aRecent[13].sSevText
    Textfield (84,326 90x19), "%s", text variable: GVL_Log.aRecent[13].sTime
    Textfield (178,326 602x19), "%s", text variable: GVL_Log.aRecent[13].sMsg
    Textfield (20,346 60x19), "%s", text variable: GVL_Log.aRecent[14].sSevText
    Textfield (84,346 90x19), "%s", text variable: GVL_Log.aRecent[14].sTime
    Textfield (178,346 602x19), "%s", text variable: GVL_Log.aRecent[14].sMsg
    Textfield (20,366 60x19), "%s", text variable: GVL_Log.aRecent[15].sSevText
    Textfield (84,366 90x19), "%s", text variable: GVL_Log.aRecent[15].sTime
    Textfield (178,366 602x19), "%s", text variable: GVL_Log.aRecent[15].sMsg
    Textfield (20,386 60x19), "%s", text variable: GVL_Log.aRecent[16].sSevText
    Textfield (84,386 90x19), "%s", text variable: GVL_Log.aRecent[16].sTime
    Textfield (178,386 602x19), "%s", text variable: GVL_Log.aRecent[16].sMsg
    Textfield (20,406 60x19), "%s", text variable: GVL_Log.aRecent[17].sSevText
    Textfield (84,406 90x19), "%s", text variable: GVL_Log.aRecent[17].sTime
    Textfield (178,406 602x19), "%s", text variable: GVL_Log.aRecent[17].sMsg
    Textfield (20,426 60x19), "%s", text variable: GVL_Log.aRecent[18].sSevText
    Textfield (84,426 90x19), "%s", text variable: GVL_Log.aRecent[18].sTime
    Textfield (178,426 602x19), "%s", text variable: GVL_Log.aRecent[18].sMsg
    Textfield (20,446 60x19), "%s", text variable: GVL_Log.aRecent[19].sSevText
    Textfield (84,446 90x19), "%s", text variable: GVL_Log.aRecent[19].sTime
    Textfield (178,446 602x19), "%s", text variable: GVL_Log.aRecent[19].sMsg
END_VISUALIZATION

// ---- VISU/Robot.TcVIS
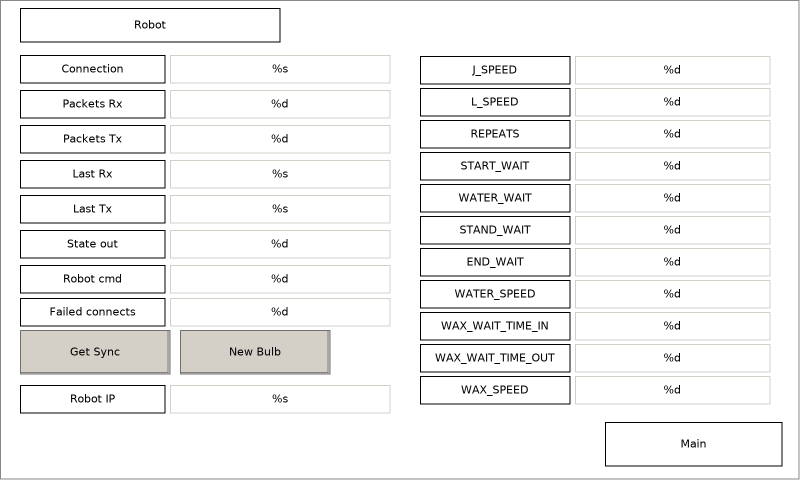
VISUALIZATION Robot  // 800x480
    Rectangle (605,422 177x44), "Main"
        OnMouseDown: change screen: Main
    Rectangle (20,8 260x34), "Robot"
    Rectangle (20,55 145x28), "Connection"
    Textfield (170,55 220x28), "%s", text variable: GVL_Robot.stRobot.sConnStateText
    Rectangle (20,90 145x28), "Packets Rx"
    Textfield (170,90 220x28), "%d", text variable: GVL_Robot.stRobot.nPacketsRx
    Rectangle (20,125 145x28), "Packets Tx"
    Textfield (170,125 220x28), "%d", text variable: GVL_Robot.stRobot.nPacketsTx
    Rectangle (20,298 145x28), "Failed connects"
    Textfield (170,298 220x28), "%d", text variable: GVL_Robot.stRobot.nConnectFails
    Rectangle (20,160 145x28), "Last Rx"
    Textfield (170,160 220x28), "%s", text variable: GVL_Robot.stRobot.sLastMessage
    Rectangle (20,195 145x28), "Last Tx"
    Textfield (170,195 220x28), "%s", text variable: GVL_Robot.stRobot.sLastTxMessage
    Rectangle (20,230 145x28), "State out"
    Textfield (170,230 220x28), "%d", text variable: GVL_Robot.stParams.nStateOut
    Rectangle (20,265 145x28), "Robot cmd"
    Textfield (170,265 220x28), "%d", text variable: GVL_Robot.stParams.nRobotCmd
    Button (20,330 150x44), "Get Sync"
        tap GVL_Robot.stParams.bGetSync
    Button (180,330 150x44), "New Bulb"
        tap GVL_Robot.stParams.bTriggerNewBulb
    Textfield (575,280 195x28), "%d", text variable: GVL_Robot.stParams.WATER_SPEED
        OnMouseClick: write the text variable via Default, min 0, max 100
    Rectangle (420,56 150x28), "J_SPEED"
    Textfield (575,56 195x28), "%d", text variable: GVL_Robot.stParams.J_SPEED
        OnMouseClick: write the text variable via Default, min 1, max 100
    Rectangle (420,88 150x28), "L_SPEED"
    Textfield (575,88 195x28), "%d", text variable: GVL_Robot.stParams.L_SPEED
        OnMouseClick: write the text variable via Default, min 1, max 100
    Rectangle (420,120 150x28), "REPEATS"
    Textfield (575,120 195x28), "%d", text variable: GVL_Robot.stParams.REPEATS
        OnMouseClick: write the text variable via Default, min 1, max 10
    Rectangle (420,152 150x28), "START_WAIT"
    Textfield (575,152 195x28), "%d", text variable: GVL_Robot.stParams.START_WAIT
        OnMouseClick: write the text variable via Default, min 10, max 10000
    Rectangle (420,184 150x28), "WATER_WAIT"
    Textfield (575,184 195x28), "%d", text variable: GVL_Robot.stParams.WATER_WAIT
        OnMouseClick: write the text variable via Default, min 10, max 10000
    Rectangle (420,216 150x28), "STAND_WAIT"
    Textfield (575,216 195x28), "%d", text variable: GVL_Robot.stParams.STAND_WAIT
        OnMouseClick: write the text variable via Default, min 10, max 10000
    Rectangle (420,248 150x28), "END_WAIT"
    Textfield (575,248 195x28), "%d", text variable: GVL_Robot.stParams.END_WAIT
        OnMouseClick: write the text variable via Default, min 10, max 10000
    Rectangle (420,280 150x28), "WATER_SPEED"
    Rectangle (420,312 150x28), "WAX_WAIT_TIME_IN"
    Textfield (575,312 195x28), "%d", text variable: GVL_Robot.stParams.WAX_WAIT_TIME_IN
        OnMouseClick: write the text variable via Default, min 0, max 10000
    Rectangle (420,344 150x28), "WAX_WAIT_TIME_OUT"
    Textfield (575,344 195x28), "%d", text variable: GVL_Robot.stParams.WAX_WAIT_TIME_OUT
        OnMouseClick: write the text variable via Default, min 10, max 10000
    Rectangle (420,376 150x28), "WAX_SPEED"
    Textfield (575,376 195x28), "%d", text variable: GVL_Robot.stParams.WAX_SPEED
        OnMouseClick: write the text variable via Default, min 0, max 100
    Rectangle (20,385 145x28), "Robot IP"
    Textfield (170,385 220x28), "%s", text variable: GVL_Robot.sRobotHost
        OnMouseClick: write the text variable via Default, title Robot IP address
END_VISUALIZATION

// ---- VISU/GripperManual.TcVIS
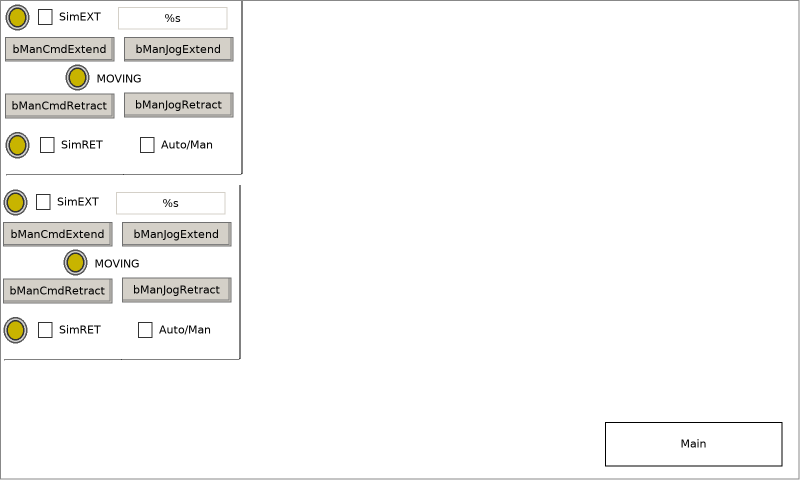
VISUALIZATION GripperManual  // 800x480
    Frame (-3,-3 250x200)
        shows Piston(piston := GVL_HMI.stGripSolL)
    Rectangle (605,422 177x44), "Main"
        OnMouseDown: change screen: Main
    Frame (-5,182 250x200)
        shows Piston(piston := GVL_HMI.stGripSolR)
END_VISUALIZATION

// ---- VISU/Piston.TcVIS
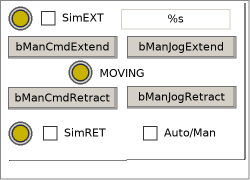
VISUALIZATION Piston  // 250x180
VAR_IN_OUT
	piston : ST_HmiPiston;
END_VAR
    Lamp1 (6,5 29x27), variable: piston.bIsExtended, style: Lamp-Lamp1-Yellow
    Button (8,36 109x22), "bManCmdExtend"
        tap piston.bManCmdExtend
    Button (127,36 109x22), "bManJogExtend"
        tap piston.bManJogExtend
    Button (127,86 109x22), "bManJogRetract"
        tap piston.bManJogRetract
    Button (8,87 109x22), "bManCmdRetract"
        tap piston.bManCmdRetract
    Textfield (121,9 109x20), "%s", text variable: piston.Name
    Lamp1 (6,120 29x27), variable: piston.bIsRetracted, style: Lamp-Lamp1-Yellow
    Label (69,62 106x23), "MOVING", invisible if: NOT(piston.bIsMoving)
    Lamp1 (66,59 29x27), variable: piston.bOutSolenoidExtend, style: Lamp-Lamp1-Yellow
    Checkbox (141,118 100x30), "Auto/Man", variable: piston.bMode
    Checkbox (41,118 84x30), "SimRET", variable: piston.bSimulateRetracted
    Checkbox (39,3 84x30), "SimEXT", variable: piston.bSimulateExtended
    Line (9,160) (244,159)
    Line (245,159) (245,3)
END_VISUALIZATION

// ---- VISU/AutoMain.TcVIS
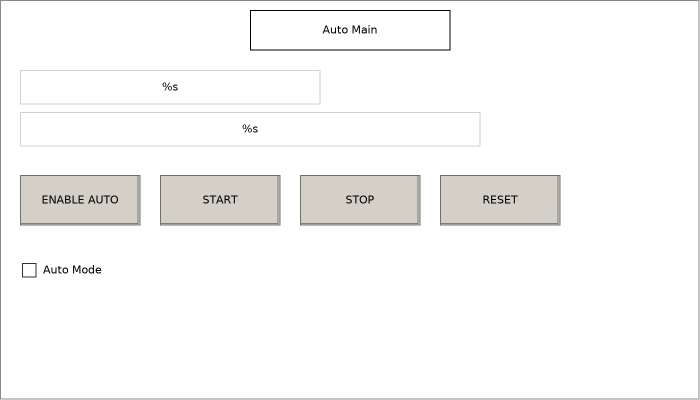
VISUALIZATION AutoMain  // 700x400
VAR_IN_OUT
	stMasterAutoCycle : ST_HmiMasterAuto;
	stCfg : ST_HmiMasterAutoCfg;
END_VAR
    Rectangle (250,10 200x40), "Auto Main"
    Textfield (20,70 300x34), "%s", text variable: stMasterAutoCycle.sStepText
    Textfield (20,112 460x34), "%s", text variable: stMasterAutoCycle.sErrorText
    Button (20,175 120x50), "ENABLE AUTO"
        tap stMasterAutoCycle.bStart
    Button (300,175 120x50), "STOP"
        tap stMasterAutoCycle.bStop
    Button (160,175 120x50), "START"
        tap stMasterAutoCycle.bStartCycle
    Button (440,175 120x50), "RESET"
        tap stMasterAutoCycle.bReset
    Checkbox (20,255 240x30), "Auto Mode", variable: GVL_HMI.bAutoMode
END_VISUALIZATION

// ---- VISU/AutoConfig.TcVIS
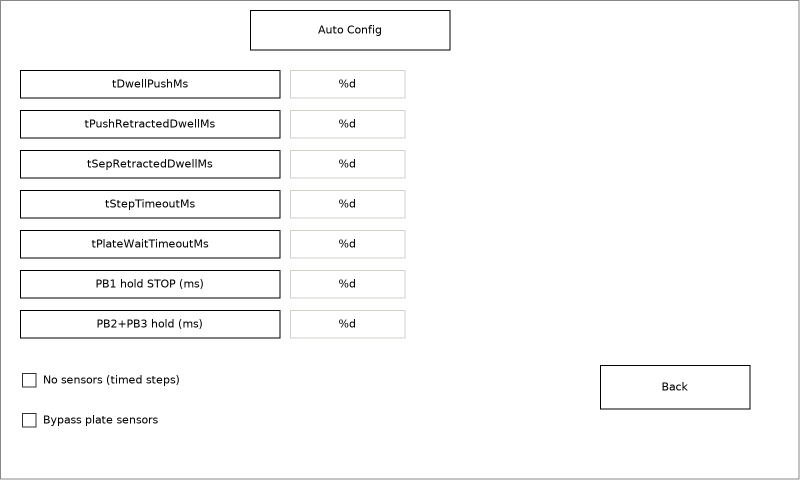
VISUALIZATION AutoConfig  // 800x480
    Rectangle (250,10 200x40), "Auto Config"
    Checkbox (20,365 240x30), "No sensors (timed steps)", variable: GVL_HmiPersistent.stMasterAutoCfg.bNoSensors
    Checkbox (20,405 240x30), "Bypass plate sensors", variable: GVL_HmiPersistent.stMasterAutoCfg.bBypassPlateSensors
    Rectangle (20,70 260x28), "tDwellPushMs"
    Textfield (290,70 115x28), "%d", text variable: GVL_HmiPersistent.stMasterAutoCfg.tDwellPushMs
        OnMouseClick: write the text variable via Default
    Rectangle (20,110 260x28), "tPushRetractedDwellMs"
    Textfield (290,110 115x28), "%d", text variable: GVL_HmiPersistent.stMasterAutoCfg.tPushRetractedDwellMs
        OnMouseClick: write the text variable via Default
    Rectangle (20,150 260x28), "tSepRetractedDwellMs"
    Textfield (290,150 115x28), "%d", text variable: GVL_HmiPersistent.stMasterAutoCfg.tSepRetractedDwellMs
        OnMouseClick: write the text variable via Default
    Rectangle (20,190 260x28), "tStepTimeoutMs"
    Textfield (290,190 115x28), "%d", text variable: GVL_HmiPersistent.stMasterAutoCfg.tStepTimeoutMs
        OnMouseClick: write the text variable via Default
    Rectangle (20,230 260x28), "tPlateWaitTimeoutMs"
    Textfield (290,230 115x28), "%d", text variable: GVL_HmiPersistent.stMasterAutoCfg.tPlateWaitTimeoutMs
        OnMouseClick: write the text variable via Default
    Rectangle (20,270 260x28), "PB1 hold STOP (ms)"
    Textfield (290,270 115x28), "%d", text variable: GVL_HmiPersistent.stMasterAutoCfg.tPbStopHoldMs
        OnMouseClick: write the text variable via Default
    Rectangle (20,310 260x28), "PB2+PB3 hold (ms)"
    Textfield (290,310 115x28), "%d", text variable: GVL_HmiPersistent.stMasterAutoCfg.tPbStartHoldMs
        OnMouseClick: write the text variable via Default
    Rectangle (600,365 150x44), "Back"
        OnMouseDown: change screen: Main
END_VISUALIZATION
